# EPICS substitutions: apps/A6551App/Db/original/userHost.substitutions
# Example substitutions file

file "db/dbExample1.db" {
    { user = "baltzellHost" }
}

file db/dbExample2.db {
    pattern { user, no, scan }
        { "baltzellHost", 1, "1 second" }
        { "baltzellHost", 2, "2 second" }
        { "baltzellHost", 3, "5 second" }
}
